(* CODESYS project FU_iMinMaxValue.xml

Project tree, tasks and I/O mapping:
  function FU_iMinMaxValue [ST]
*)

// FU_iMinMaxValue
//This function keeps a variable between a minimum and a maximum value
// +-----------+----------+----------+-----------------------------------------------------------------------------------------------------------------------+
// |**Version**|**Author**| **Date** |**Changes**                                                                                                            |
// +-----------+----------+----------+-----------------------------------------------------------------------------------------------------------------------+
// | 1         | NSN      | 07-01-18 | Creation                                                                                                              |
// +-----------+----------+----------+-----------------------------------------------------------------------------------------------------------------------+
FUNCTION FU_iMinMaxValue : BOOL
VAR_IN_OUT
	Variable		:INT;
END_VAR
VAR_INPUT
	MinVal			:INT;
	MaxVal			:INT;
END_VAR

IF Variable < MinVal THEN			//This makes sure only values between 0 and 10000 can be entered
	Variable				:=		MinVal;
ELSIF Variable > MaxVal THEN
	Variable				:=		MaxVal;
END_IF

END_FUNCTION
